Staubli VAL3: N22_PosDosi.pgx

program N22_PosDosi()
  local pointRx l_pDosi
begin

  // Moure puntes per treure les gotes
  l_pDosi=here(tToolActiva,fTaula)
  l_pDosi.trsf.x=l_pDosi.trsf.x+nXOffset
  l_pDosi.trsf.y=l_pDosi.trsf.y+nYOffset
  l_pDosi.trsf.z=l_pDosi.trsf.z+nZOffset
  movel(l_pDosi,tToolActiva,mLent)
  waitEndMove()

  bTaskDone=true
end
